FUNCTION_BLOCK GF_Warten EXTENDS FB_Basisfunktionalitaeten
VAR_INPUT
	// Instanzieren von Sensoren mit Interfaces
	
	// Instanzieren von Aktoren mit Interfaces
	
END_VAR
VAR_OUTPUT
	
END_VAR
VAR
	
END_VAR

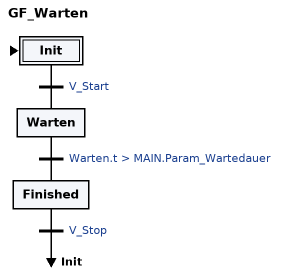
INITIAL_STEP Init:
END_STEP
TRANSITION FROM Init TO Warten
    := V_Start;
END_TRANSITION
STEP Warten:
END_STEP
TRANSITION FROM Warten TO Finished
    := Warten.t > MAIN.Param_Wartedauer;
END_TRANSITION
STEP Finished:
END_STEP
TRANSITION FROM Finished TO Init
    := V_Stop;
END_TRANSITION

END_FUNCTION_BLOCK

(* stored: Version 1.1.0.1, ProductVersion 3.1.4024.12
   POU GF_Warten: Id {3b1967cc-b232-47bd-a538-3325a138e01c}, SpecialFunc None *)
